// TIA Portal V17 export
// export: Created 2022-03-12T16:05:15.6191488Z, ExportSetting WithDefaults, DisplayName Totally Integrated Automation Portal, DisplayVersion V17, DisplayName TIA Portal Openness, DisplayVersion V17, DisplayName TIA Portal Version Control Interface, DisplayVersion V17, DisplayName STEP 7 Professional, DisplayVersion V17, DisplayName STEP 7 Safety, DisplayVersion V17, DisplayName WinCC Advanced / Unified PC, DisplayVersion V17
FUNCTION_BLOCK "UN_07_RecipeControl"   // FB31627, LAD
TITLE = UN_07_RecipeControl
{ S7_Optimized_Access := 'TRUE' }
AUTHOR : tech.team.motioncontrol@siemens.com
FAMILY : CPG
VERSION : 1.0
// Support: tech.team.motioncontrol@siemens.com
// stored: AutoNumber true, IsIECCheckEnabled false, IsRetainMemResEnabled false, MemoryReserve 100, SetENOAutomatically false, UDAEnableTagReadback false
   VAR
      instRecipeControl { ExternalAccessible := 'False'; ExternalVisible := 'False'; ExternalWritable := 'False'; S7_SetPoint := 'True'} : "CPG_RecipeControl";
      instRecipeManager { ExternalAccessible := 'False'; ExternalVisible := 'False'; ExternalWritable := 'False'; S7_SetPoint := 'True'} : "CPG_RecipeHMIManager";
      ONS_RecipeChange { ExternalAccessible := 'False'; ExternalVisible := 'False'; ExternalWritable := 'False'} : Bool;
      ONS_SaveAsChange { ExternalAccessible := 'False'; ExternalVisible := 'False'; ExternalWritable := 'False'} : Bool;
      ONS_DeleteChange { ExternalAccessible := 'False'; ExternalVisible := 'False'; ExternalWritable := 'False'} : Bool;
      ONS_CopyChange { ExternalAccessible := 'False'; ExternalVisible := 'False'; ExternalWritable := 'False'} : Bool;
   END_VAR
   VAR_TEMP
      tempEnablechange : Bool;
      tempRecipenewname : String[60];
      tempErrorID : Word;
      tempError : Word;
      tempSeconds : Time;
   END_VAR
   VAR CONSTANT
      ERR_CHANGE : Word := 16#8001;
      ERR_SAVE : Word := 16#8002;
      ERR_COPY : Word := 16#8004;
      ERR_DELETE : Word := 16#8008;
   END_VAR
   VAR_TEMP   // added for the SCL form of the ladder/FBD networks
      _w1 : Bool;
      _w2 : Bool;
   END_VAR
BEGIN

REGION Network 1: Determine if recipe change is permitted based on machine state
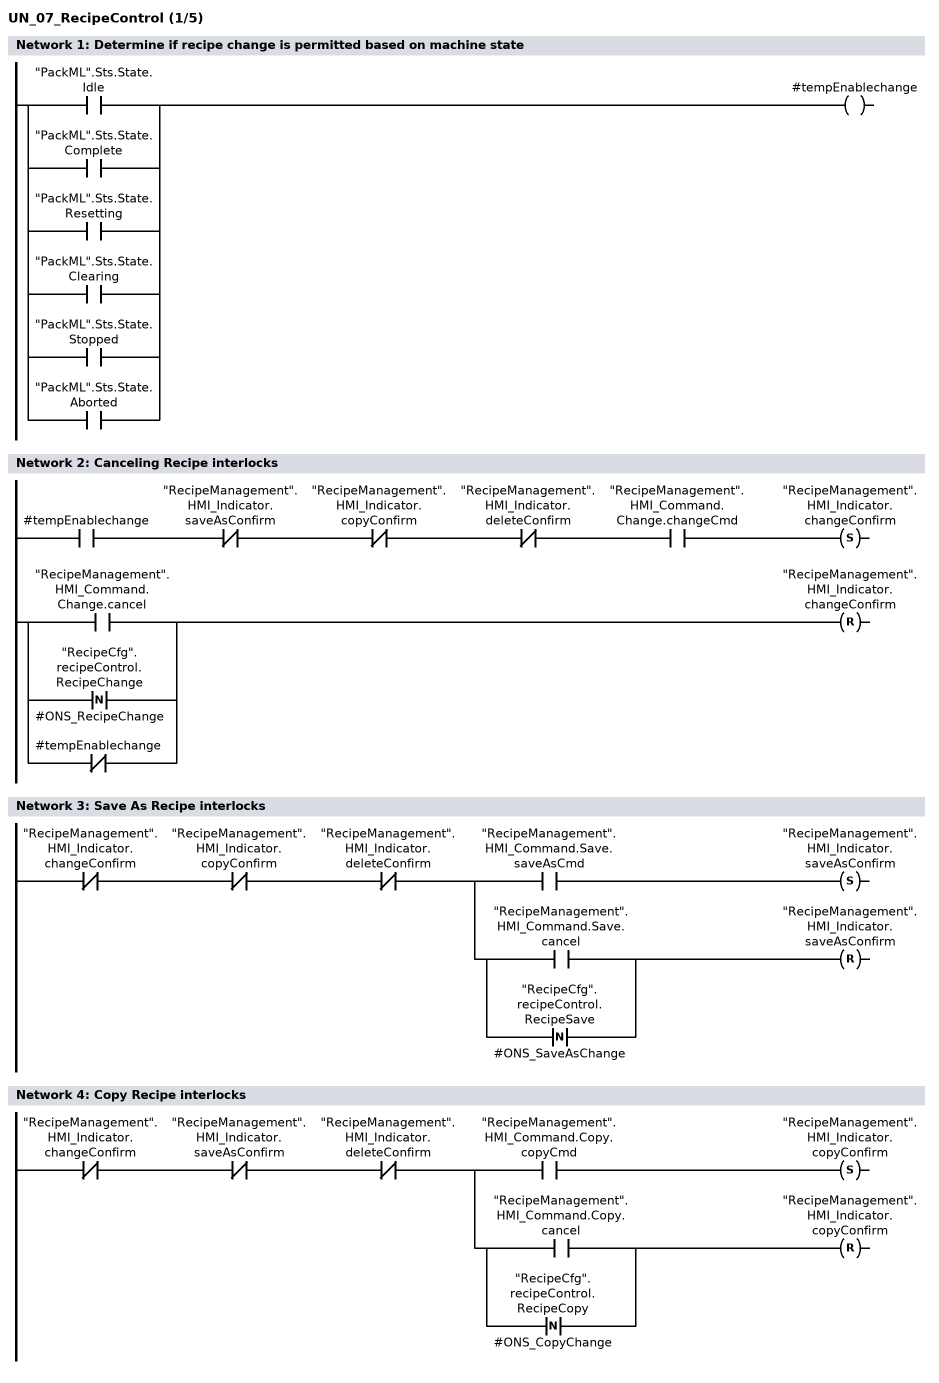
   RUNG wire#powerrail
      Contact( "PackML".Sts.State.Idle )
      wire#w1
      Coil( #tempEnablechange )
   END_RUNG
   RUNG wire#powerrail
      Contact( "PackML".Sts.State.Complete )
   END_RUNG wire#w1
   RUNG wire#powerrail
      Contact( "PackML".Sts.State.Resetting )
   END_RUNG wire#w1
   RUNG wire#powerrail
      Contact( "PackML".Sts.State.Clearing )
   END_RUNG wire#w1
   RUNG wire#powerrail
      Contact( "PackML".Sts.State.Stopped )
   END_RUNG wire#w1
   RUNG wire#powerrail
      Contact( "PackML".Sts.State.Aborted )
   END_RUNG wire#w1
   // the same network as SCL:
   #tempEnablechange := "PackML".Sts.State.Idle OR "PackML".Sts.State.Complete OR "PackML".Sts.State.Resetting OR "PackML".Sts.State.Clearing OR "PackML".Sts.State.Stopped OR "PackML".Sts.State.Aborted;
END_REGION

REGION Network 2: Canceling Recipe interlocks
   RUNG wire#powerrail
      Contact( #tempEnablechange )
      I_Contact( "RecipeManagement".HMI_Indicator.saveAsConfirm )
      I_Contact( "RecipeManagement".HMI_Indicator.copyConfirm )
      I_Contact( "RecipeManagement".HMI_Indicator.deleteConfirm )
      Contact( "RecipeManagement".HMI_Command.Change.changeCmd )
      S_Coil( "RecipeManagement".HMI_Indicator.changeConfirm )
   END_RUNG
   RUNG wire#powerrail
      Contact( "RecipeManagement".HMI_Command.Change.cancel )
      wire#w1
      R_Coil( "RecipeManagement".HMI_Indicator.changeConfirm )
   END_RUNG
   RUNG wire#powerrail
      N_Contact(operand := "RecipeCfg".recipeControl.RecipeChange, bit := #ONS_RecipeChange)
   END_RUNG wire#w1
   RUNG wire#powerrail
      I_Contact( #tempEnablechange )
   END_RUNG wire#w1
   // the same network as SCL:
   IF #tempEnablechange AND NOT "RecipeManagement".HMI_Indicator.saveAsConfirm AND NOT "RecipeManagement".HMI_Indicator.copyConfirm AND NOT "RecipeManagement".HMI_Indicator.deleteConfirm AND "RecipeManagement".HMI_Command.Change.changeCmd THEN
       "RecipeManagement".HMI_Indicator.changeConfirm := TRUE;
   END_IF;
   #_w1 := NOT "RecipeCfg".recipeControl.RecipeChange AND #ONS_RecipeChange;   // falling edge of "RecipeCfg".recipeControl.RecipeChange
   #ONS_RecipeChange := "RecipeCfg".recipeControl.RecipeChange;
   IF "RecipeManagement".HMI_Command.Change.cancel OR #_w1 OR NOT #tempEnablechange THEN
       "RecipeManagement".HMI_Indicator.changeConfirm := FALSE;
   END_IF;
END_REGION

REGION Network 3: Save As Recipe interlocks
   RUNG wire#powerrail
      I_Contact( "RecipeManagement".HMI_Indicator.changeConfirm )
      I_Contact( "RecipeManagement".HMI_Indicator.copyConfirm )
      I_Contact( "RecipeManagement".HMI_Indicator.deleteConfirm )
      wire#w1
      Contact( "RecipeManagement".HMI_Command.Save.saveAsCmd )
      S_Coil( "RecipeManagement".HMI_Indicator.saveAsConfirm )
   END_RUNG
   RUNG wire#w1
      Contact( "RecipeManagement".HMI_Command.Save.cancel )
      wire#w2
      R_Coil( "RecipeManagement".HMI_Indicator.saveAsConfirm )
   END_RUNG
   RUNG wire#w1
      N_Contact(operand := "RecipeCfg".recipeControl.RecipeSave, bit := #ONS_SaveAsChange)
   END_RUNG wire#w2
   // the same network as SCL:
   #_w1 := NOT "RecipeManagement".HMI_Indicator.changeConfirm AND NOT "RecipeManagement".HMI_Indicator.copyConfirm AND NOT "RecipeManagement".HMI_Indicator.deleteConfirm;
   IF #_w1 AND "RecipeManagement".HMI_Command.Save.saveAsCmd THEN
       "RecipeManagement".HMI_Indicator.saveAsConfirm := TRUE;
   END_IF;
   #_w2 := #_w1 AND NOT "RecipeCfg".recipeControl.RecipeSave AND #ONS_SaveAsChange;   // falling edge of "RecipeCfg".recipeControl.RecipeSave
   #ONS_SaveAsChange := "RecipeCfg".recipeControl.RecipeSave;
   IF (#_w1 AND "RecipeManagement".HMI_Command.Save.cancel) OR #_w2 THEN
       "RecipeManagement".HMI_Indicator.saveAsConfirm := FALSE;
   END_IF;
END_REGION

REGION Network 4: Copy Recipe interlocks
   RUNG wire#powerrail
      I_Contact( "RecipeManagement".HMI_Indicator.changeConfirm )
      I_Contact( "RecipeManagement".HMI_Indicator.saveAsConfirm )
      I_Contact( "RecipeManagement".HMI_Indicator.deleteConfirm )
      wire#w1
      Contact( "RecipeManagement".HMI_Command.Copy.copyCmd )
      S_Coil( "RecipeManagement".HMI_Indicator.copyConfirm )
   END_RUNG
   RUNG wire#w1
      Contact( "RecipeManagement".HMI_Command.Copy.cancel )
      wire#w2
      R_Coil( "RecipeManagement".HMI_Indicator.copyConfirm )
   END_RUNG
   RUNG wire#w1
      N_Contact(operand := "RecipeCfg".recipeControl.RecipeCopy, bit := #ONS_CopyChange)
   END_RUNG wire#w2
   // the same network as SCL:
   #_w1 := NOT "RecipeManagement".HMI_Indicator.changeConfirm AND NOT "RecipeManagement".HMI_Indicator.saveAsConfirm AND NOT "RecipeManagement".HMI_Indicator.deleteConfirm;
   IF #_w1 AND "RecipeManagement".HMI_Command.Copy.copyCmd THEN
       "RecipeManagement".HMI_Indicator.copyConfirm := TRUE;
   END_IF;
   #_w2 := #_w1 AND NOT "RecipeCfg".recipeControl.RecipeCopy AND #ONS_CopyChange;   // falling edge of "RecipeCfg".recipeControl.RecipeCopy
   #ONS_CopyChange := "RecipeCfg".recipeControl.RecipeCopy;
   IF (#_w1 AND "RecipeManagement".HMI_Command.Copy.cancel) OR #_w2 THEN
       "RecipeManagement".HMI_Indicator.copyConfirm := FALSE;
   END_IF;
END_REGION

REGION Network 5: Delete Recipe interlocks
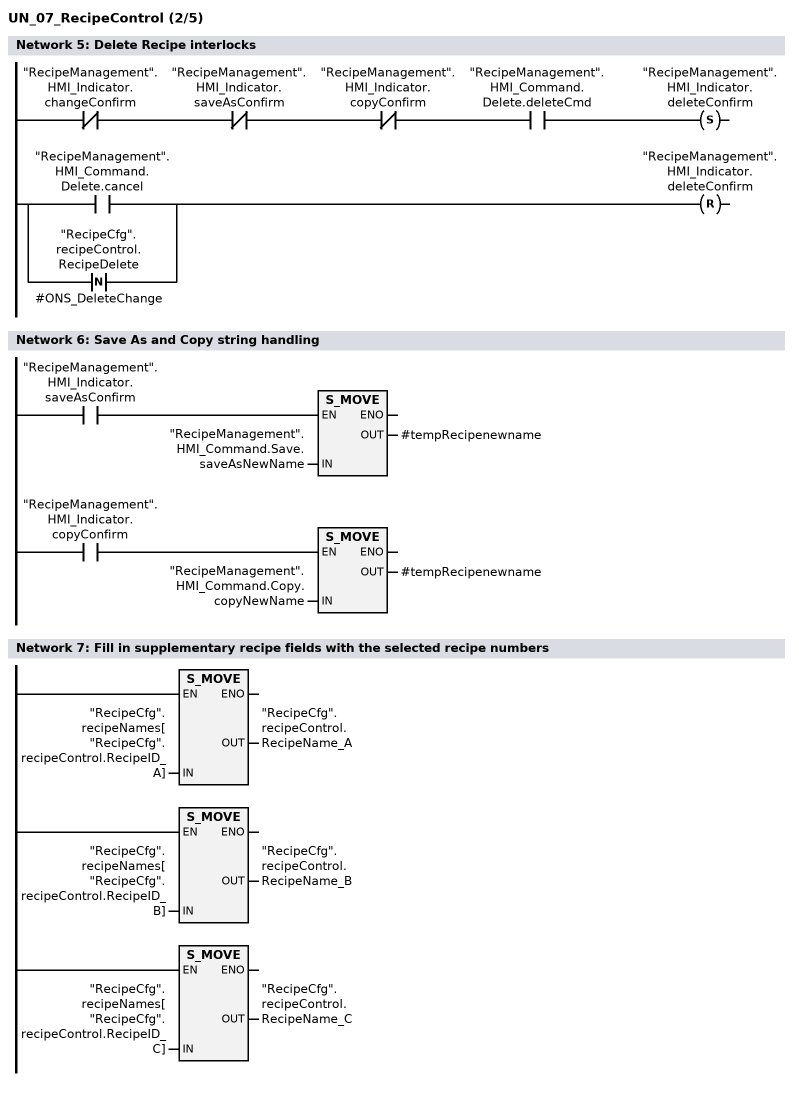
   RUNG wire#powerrail
      I_Contact( "RecipeManagement".HMI_Indicator.changeConfirm )
      I_Contact( "RecipeManagement".HMI_Indicator.saveAsConfirm )
      I_Contact( "RecipeManagement".HMI_Indicator.copyConfirm )
      Contact( "RecipeManagement".HMI_Command.Delete.deleteCmd )
      S_Coil( "RecipeManagement".HMI_Indicator.deleteConfirm )
   END_RUNG
   RUNG wire#powerrail
      Contact( "RecipeManagement".HMI_Command.Delete.cancel )
      wire#w1
      R_Coil( "RecipeManagement".HMI_Indicator.deleteConfirm )
   END_RUNG
   RUNG wire#powerrail
      N_Contact(operand := "RecipeCfg".recipeControl.RecipeDelete, bit := #ONS_DeleteChange)
   END_RUNG wire#w1
   // the same network as SCL:
   IF NOT "RecipeManagement".HMI_Indicator.changeConfirm AND NOT "RecipeManagement".HMI_Indicator.saveAsConfirm AND NOT "RecipeManagement".HMI_Indicator.copyConfirm AND "RecipeManagement".HMI_Command.Delete.deleteCmd THEN
       "RecipeManagement".HMI_Indicator.deleteConfirm := TRUE;
   END_IF;
   #_w1 := NOT "RecipeCfg".recipeControl.RecipeDelete AND #ONS_DeleteChange;   // falling edge of "RecipeCfg".recipeControl.RecipeDelete
   #ONS_DeleteChange := "RecipeCfg".recipeControl.RecipeDelete;
   IF "RecipeManagement".HMI_Command.Delete.cancel OR #_w1 THEN
       "RecipeManagement".HMI_Indicator.deleteConfirm := FALSE;
   END_IF;
END_REGION

REGION Network 6: Save As and Copy string handling
   RUNG wire#powerrail
      Contact( "RecipeManagement".HMI_Indicator.saveAsConfirm )
      S_Move(in := "RecipeManagement".HMI_Command.Save.saveAsNewName, out => #tempRecipenewname)
   END_RUNG
   RUNG wire#powerrail
      Contact( "RecipeManagement".HMI_Indicator.copyConfirm )
      S_Move(in := "RecipeManagement".HMI_Command.Copy.copyNewName, out => #tempRecipenewname)
   END_RUNG
   // the same network as SCL:
   IF "RecipeManagement".HMI_Indicator.saveAsConfirm THEN
       #tempRecipenewname := "RecipeManagement".HMI_Command.Save.saveAsNewName;
   END_IF;
   IF "RecipeManagement".HMI_Indicator.copyConfirm THEN
       #tempRecipenewname := "RecipeManagement".HMI_Command.Copy.copyNewName;
   END_IF;
END_REGION

REGION Network 7: Fill in supplementary recipe fields with the selected recipe numbers
   RUNG wire#powerrail
      S_Move(in := "RecipeCfg".recipeNames["RecipeCfg".recipeControl.RecipeID_A], out => "RecipeCfg".recipeControl.RecipeName_A)
   END_RUNG
   RUNG wire#powerrail
      S_Move(in := "RecipeCfg".recipeNames["RecipeCfg".recipeControl.RecipeID_B], out => "RecipeCfg".recipeControl.RecipeName_B)
   END_RUNG
   RUNG wire#powerrail
      S_Move(in := "RecipeCfg".recipeNames["RecipeCfg".recipeControl.RecipeID_C], out => "RecipeCfg".recipeControl.RecipeName_C)
   END_RUNG
   // the same network as SCL:
   "RecipeCfg".recipeControl.RecipeName_A := "RecipeCfg".recipeNames["RecipeCfg".recipeControl.RecipeID_A];
   "RecipeCfg".recipeControl.RecipeName_B := "RecipeCfg".recipeNames["RecipeCfg".recipeControl.RecipeID_B];
   "RecipeCfg".recipeControl.RecipeName_C := "RecipeCfg".recipeNames["RecipeCfg".recipeControl.RecipeID_C];
END_REGION

REGION Network 8: Call Recipe Control
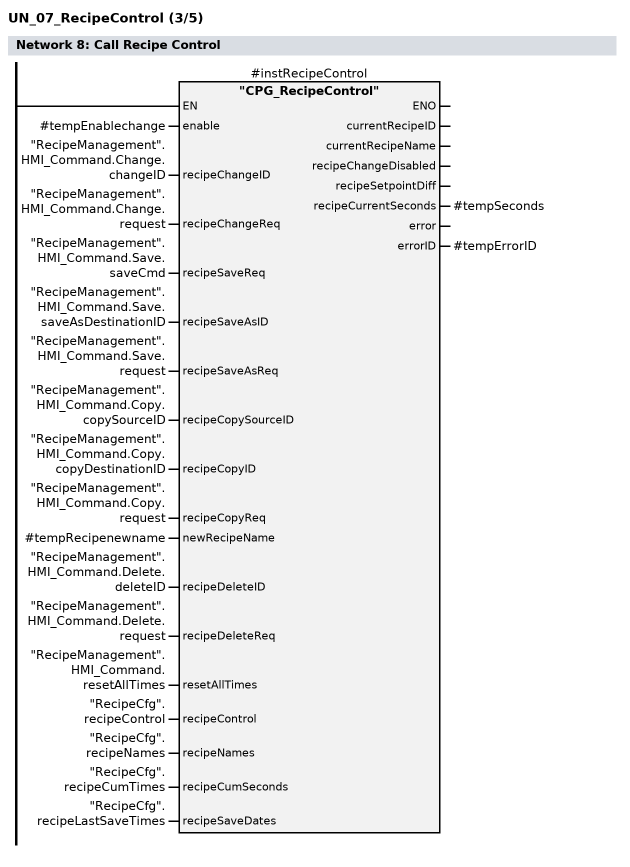
   RUNG wire#powerrail
      #instRecipeControl(enable := #tempEnablechange, recipeChangeID := "RecipeManagement".HMI_Command.Change.changeID, recipeChangeReq := "RecipeManagement".HMI_Command.Change.request, recipeSaveReq := "RecipeManagement".HMI_Command.Save.saveCmd, recipeSaveAsID := "RecipeManagement".HMI_Command.Save.saveAsDestinationID, recipeSaveAsReq := "RecipeManagement".HMI_Command.Save.request, recipeCopySourceID := "RecipeManagement".HMI_Command.Copy.copySourceID, recipeCopyID := "RecipeManagement".HMI_Command.Copy.copyDestinationID, recipeCopyReq := "RecipeManagement".HMI_Command.Copy.request, newRecipeName := #tempRecipenewname, recipeDeleteID := "RecipeManagement".HMI_Command.Delete.deleteID, recipeDeleteReq := "RecipeManagement".HMI_Command.Delete.request, resetAllTimes := "RecipeManagement".HMI_Command.resetAllTimes, recipeControl := "RecipeCfg".recipeControl, recipeNames := "RecipeCfg".recipeNames, recipeCumSeconds := "RecipeCfg".recipeCumTimes, recipeSaveDates := "RecipeCfg".recipeLastSaveTimes, currentRecipeID =>, currentRecipeName =>, recipeChangeDisabled =>, recipeSetpointDiff =>, recipeCurrentSeconds => #tempSeconds, error =>, errorID => #tempErrorID)
   END_RUNG
   // the same network as SCL:
   #instRecipeControl(enable := #tempEnablechange,   // "CPG_RecipeControl"
                      recipeChangeID := "RecipeManagement".HMI_Command.Change.changeID,
                      recipeChangeReq := "RecipeManagement".HMI_Command.Change.request,
                      recipeSaveReq := "RecipeManagement".HMI_Command.Save.saveCmd,
                      recipeSaveAsID := "RecipeManagement".HMI_Command.Save.saveAsDestinationID,
                      recipeSaveAsReq := "RecipeManagement".HMI_Command.Save.request,
                      recipeCopySourceID := "RecipeManagement".HMI_Command.Copy.copySourceID,
                      recipeCopyID := "RecipeManagement".HMI_Command.Copy.copyDestinationID,
                      recipeCopyReq := "RecipeManagement".HMI_Command.Copy.request,
                      newRecipeName := #tempRecipenewname,
                      recipeDeleteID := "RecipeManagement".HMI_Command.Delete.deleteID,
                      recipeDeleteReq := "RecipeManagement".HMI_Command.Delete.request,
                      resetAllTimes := "RecipeManagement".HMI_Command.resetAllTimes,
                      recipeControl := "RecipeCfg".recipeControl,
                      recipeNames := "RecipeCfg".recipeNames,
                      recipeCumSeconds := "RecipeCfg".recipeCumTimes,
                      recipeSaveDates := "RecipeCfg".recipeLastSaveTimes,
                      recipeCurrentSeconds => #tempSeconds,
                      errorID => #tempErrorID);
END_REGION

REGION Network 9: Clear IDs from HMI if not on that screen
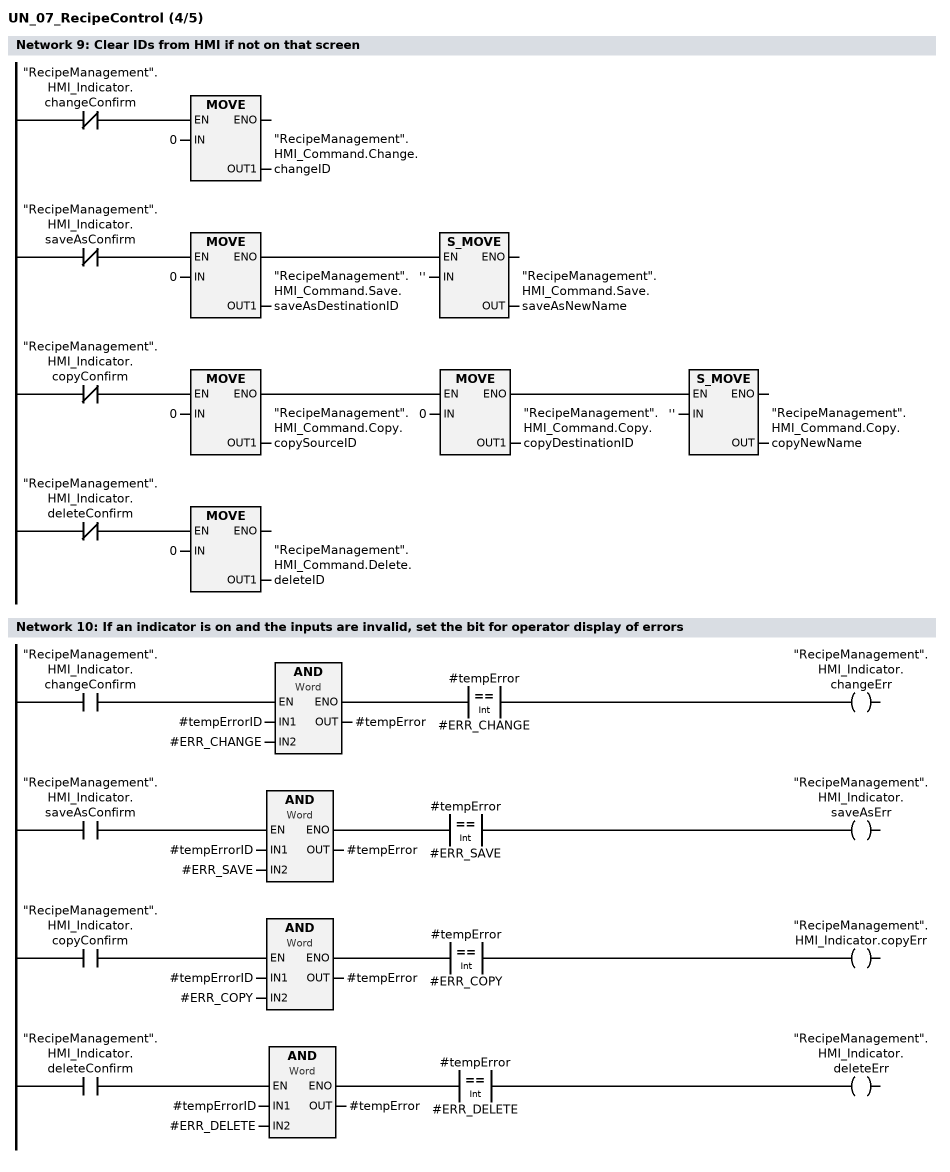
   RUNG wire#powerrail
      I_Contact( "RecipeManagement".HMI_Indicator.changeConfirm )
      Move(in := 0, out1 => "RecipeManagement".HMI_Command.Change.changeID)
   END_RUNG
   RUNG wire#powerrail
      I_Contact( "RecipeManagement".HMI_Indicator.saveAsConfirm )
      Move(in := 0, out1 => "RecipeManagement".HMI_Command.Save.saveAsDestinationID)
      S_Move(in := '', out => "RecipeManagement".HMI_Command.Save.saveAsNewName)
   END_RUNG
   RUNG wire#powerrail
      I_Contact( "RecipeManagement".HMI_Indicator.copyConfirm )
      Move(in := 0, out1 => "RecipeManagement".HMI_Command.Copy.copySourceID)
      Move(in := 0, out1 => "RecipeManagement".HMI_Command.Copy.copyDestinationID)
      S_Move(in := '', out => "RecipeManagement".HMI_Command.Copy.copyNewName)
   END_RUNG
   RUNG wire#powerrail
      I_Contact( "RecipeManagement".HMI_Indicator.deleteConfirm )
      Move(in := 0, out1 => "RecipeManagement".HMI_Command.Delete.deleteID)
   END_RUNG
   // the same network as SCL:
   IF NOT "RecipeManagement".HMI_Indicator.changeConfirm THEN
       "RecipeManagement".HMI_Command.Change.changeID := 0;
   END_IF;
   IF NOT "RecipeManagement".HMI_Indicator.saveAsConfirm THEN
       "RecipeManagement".HMI_Command.Save.saveAsDestinationID := 0;
       "RecipeManagement".HMI_Command.Save.saveAsNewName := '';
   END_IF;
   IF NOT "RecipeManagement".HMI_Indicator.copyConfirm THEN
       "RecipeManagement".HMI_Command.Copy.copySourceID := 0;
       "RecipeManagement".HMI_Command.Copy.copyDestinationID := 0;
       "RecipeManagement".HMI_Command.Copy.copyNewName := '';
   END_IF;
   IF NOT "RecipeManagement".HMI_Indicator.deleteConfirm THEN
       "RecipeManagement".HMI_Command.Delete.deleteID := 0;
   END_IF;
END_REGION

REGION Network 10: If an indicator is on and the inputs are invalid, set the bit for operator display of errors
   RUNG wire#powerrail
      Contact( "RecipeManagement".HMI_Indicator.changeConfirm )
      { S7_Templates := "SrcType := Word" } And(in1 := #tempErrorID, in2 := #ERR_CHANGE, out => #tempError)
      { S7_Templates := "SrcType := Int" } EQ_Contact(in1 := #tempError, in2 := #ERR_CHANGE)
      Coil( "RecipeManagement".HMI_Indicator.changeErr )
   END_RUNG
   RUNG wire#powerrail
      Contact( "RecipeManagement".HMI_Indicator.saveAsConfirm )
      { S7_Templates := "SrcType := Word" } And(in1 := #tempErrorID, in2 := #ERR_SAVE, out => #tempError)
      { S7_Templates := "SrcType := Int" } EQ_Contact(in1 := #tempError, in2 := #ERR_SAVE)
      Coil( "RecipeManagement".HMI_Indicator.saveAsErr )
   END_RUNG
   RUNG wire#powerrail
      Contact( "RecipeManagement".HMI_Indicator.copyConfirm )
      { S7_Templates := "SrcType := Word" } And(in1 := #tempErrorID, in2 := #ERR_COPY, out => #tempError)
      { S7_Templates := "SrcType := Int" } EQ_Contact(in1 := #tempError, in2 := #ERR_COPY)
      Coil( "RecipeManagement".HMI_Indicator.copyErr )
   END_RUNG
   RUNG wire#powerrail
      Contact( "RecipeManagement".HMI_Indicator.deleteConfirm )
      { S7_Templates := "SrcType := Word" } And(in1 := #tempErrorID, in2 := #ERR_DELETE, out => #tempError)
      { S7_Templates := "SrcType := Int" } EQ_Contact(in1 := #tempError, in2 := #ERR_DELETE)
      Coil( "RecipeManagement".HMI_Indicator.deleteErr )
   END_RUNG
   // the same network as SCL:
   IF "RecipeManagement".HMI_Indicator.changeConfirm THEN #tempError := #tempErrorID AND #ERR_CHANGE; END_IF;
   "RecipeManagement".HMI_Indicator.changeErr := "RecipeManagement".HMI_Indicator.changeConfirm AND (#tempError = #ERR_CHANGE);
   IF "RecipeManagement".HMI_Indicator.saveAsConfirm THEN #tempError := #tempErrorID AND #ERR_SAVE; END_IF;
   "RecipeManagement".HMI_Indicator.saveAsErr := "RecipeManagement".HMI_Indicator.saveAsConfirm AND (#tempError = #ERR_SAVE);
   IF "RecipeManagement".HMI_Indicator.copyConfirm THEN #tempError := #tempErrorID AND #ERR_COPY; END_IF;
   "RecipeManagement".HMI_Indicator.copyErr := "RecipeManagement".HMI_Indicator.copyConfirm AND (#tempError = #ERR_COPY);
   IF "RecipeManagement".HMI_Indicator.deleteConfirm THEN #tempError := #tempErrorID AND #ERR_DELETE; END_IF;
   "RecipeManagement".HMI_Indicator.deleteErr := "RecipeManagement".HMI_Indicator.deleteConfirm AND (#tempError = #ERR_DELETE);
END_REGION

REGION Network 11: Call Recipe HMI Manager to handle display of setpoints
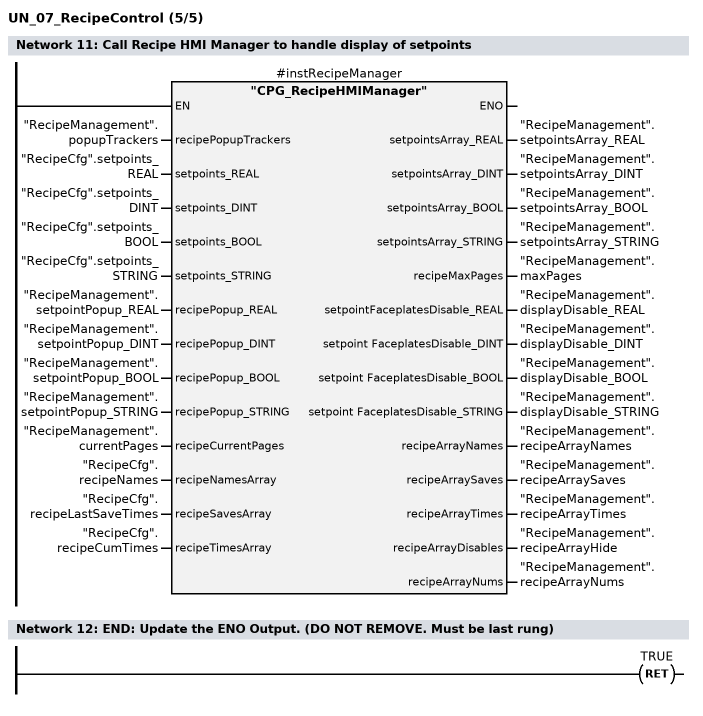
   RUNG wire#powerrail
      #instRecipeManager(recipePopupTrackers := "RecipeManagement".popupTrackers, setpoints_REAL := "RecipeCfg".setpoints_REAL, setpoints_DINT := "RecipeCfg".setpoints_DINT, setpoints_BOOL := "RecipeCfg".setpoints_BOOL, setpoints_STRING := "RecipeCfg".setpoints_STRING, recipePopup_REAL := "RecipeManagement".setpointPopup_REAL, recipePopup_DINT := "RecipeManagement".setpointPopup_DINT, recipePopup_BOOL := "RecipeManagement".setpointPopup_BOOL, recipePopup_STRING := "RecipeManagement".setpointPopup_STRING, recipeCurrentPages := "RecipeManagement".currentPages, recipeNamesArray := "RecipeCfg".recipeNames, recipeSavesArray := "RecipeCfg".recipeLastSaveTimes, recipeTimesArray := "RecipeCfg".recipeCumTimes, setpointsArray_REAL => "RecipeManagement".setpointsArray_REAL, setpointsArray_DINT => "RecipeManagement".setpointsArray_DINT, setpointsArray_BOOL => "RecipeManagement".setpointsArray_BOOL, setpointsArray_STRING => "RecipeManagement".setpointsArray_STRING, recipeMaxPages => "RecipeManagement".maxPages, setpointFaceplatesDisable_REAL => "RecipeManagement".displayDisable_REAL, "setpoint FaceplatesDisable_DINT" => "RecipeManagement".displayDisable_DINT, "setpoint FaceplatesDisable_BOOL" => "RecipeManagement".displayDisable_BOOL, "setpoint FaceplatesDisable_STRING" => "RecipeManagement".displayDisable_STRING, recipeArrayNames => "RecipeManagement".recipeArrayNames, recipeArraySaves => "RecipeManagement".recipeArraySaves, recipeArrayTimes => "RecipeManagement".recipeArrayTimes, recipeArrayDisables => "RecipeManagement".recipeArrayHide, recipeArrayNums => "RecipeManagement".recipeArrayNums)
   END_RUNG
   // the same network as SCL:
   #instRecipeManager(recipePopupTrackers := "RecipeManagement".popupTrackers,   // "CPG_RecipeHMIManager"
                      setpoints_REAL := "RecipeCfg".setpoints_REAL,
                      setpoints_DINT := "RecipeCfg".setpoints_DINT,
                      setpoints_BOOL := "RecipeCfg".setpoints_BOOL,
                      setpoints_STRING := "RecipeCfg".setpoints_STRING,
                      recipePopup_REAL := "RecipeManagement".setpointPopup_REAL,
                      recipePopup_DINT := "RecipeManagement".setpointPopup_DINT,
                      recipePopup_BOOL := "RecipeManagement".setpointPopup_BOOL,
                      recipePopup_STRING := "RecipeManagement".setpointPopup_STRING,
                      recipeCurrentPages := "RecipeManagement".currentPages,
                      recipeNamesArray := "RecipeCfg".recipeNames,
                      recipeSavesArray := "RecipeCfg".recipeLastSaveTimes,
                      recipeTimesArray := "RecipeCfg".recipeCumTimes,
                      setpointsArray_REAL => "RecipeManagement".setpointsArray_REAL,
                      setpointsArray_DINT => "RecipeManagement".setpointsArray_DINT,
                      setpointsArray_BOOL => "RecipeManagement".setpointsArray_BOOL,
                      setpointsArray_STRING => "RecipeManagement".setpointsArray_STRING,
                      recipeMaxPages => "RecipeManagement".maxPages,
                      setpointFaceplatesDisable_REAL => "RecipeManagement".displayDisable_REAL,
                      "setpoint FaceplatesDisable_DINT" => "RecipeManagement".displayDisable_DINT,
                      "setpoint FaceplatesDisable_BOOL" => "RecipeManagement".displayDisable_BOOL,
                      "setpoint FaceplatesDisable_STRING" => "RecipeManagement".displayDisable_STRING,
                      recipeArrayNames => "RecipeManagement".recipeArrayNames,
                      recipeArraySaves => "RecipeManagement".recipeArraySaves,
                      recipeArrayTimes => "RecipeManagement".recipeArrayTimes,
                      recipeArrayDisables => "RecipeManagement".recipeArrayHide,
                      recipeArrayNums => "RecipeManagement".recipeArrayNums);
END_REGION

REGION Network 12: END: Update the ENO Output. (DO NOT REMOVE. Must be last rung)
   RUNG wire#powerrail
      ReturnCoil( TRUE )
   END_RUNG
   // the same network as SCL:
   ENO := TRUE;
   RETURN;
END_REGION
END_FUNCTION_BLOCK
